{attribute 'qualified_only'}
{attribute 'strict'}
{attribute 'to_string'}
TYPE M1Detection :
(
	Read,
	ReadBuffer,
	Analyze,
	Write,
	WriteBuffer,
	Done,
	Error
	
);
END_TYPE

(* stored: Version 1.1.0.1, ProductVersion 3.1.4026.8
   DUT M1Detection: Id {e5e14681-eb87-0137-0ee9-7067820e8cb5} *)
